FUNCTION fnLogMsg : BOOL
VAR_INPUT
		logMsgPtr : POINTER TO LogMsg;
		messageLevel : enumLogMessageLevelSeverity;
		textMessage : STRING[LOG_MSG_TEXT_LENGTH];
		param1 : DINT;
		param2 : DINT;
		param3 : DINT;
END_VAR

fnLogMsg := logMsgPtr^.LogMsg(messageLevel, textMessage, param1, param2, param3, 0, 0, 0);

END_FUNCTION

(* stored: Version 1.1.0.1, ProductVersion 3.1.4024.3
   POU fnLogMsg: Id {94da9246-4759-0589-108e-6a38022822df}, SpecialFunc None *)
